// TIA Portal V18 export
// export: Created 2026-06-08T16:32:21.4329296Z, ExportSetting WithDefaults, DisplayName Totally Integrated Automation Portal, DisplayVersion V18, DisplayName TIA Portal Openness, DisplayVersion V18, DisplayName TIA Portal Version Control Interface, DisplayVersion V18, DisplayName STEP 7 Professional, DisplayVersion V18, DisplayName STEP 7 Safety, DisplayVersion V18, DisplayName WinCC Professional, DisplayVersion V18
FUNCTION_BLOCK "Assembly_Blue"   // FB11, LAD
VERSION : 0.1
// stored: AutoNumber true, IsIECCheckEnabled false, UDAEnableTagReadback false
   VAR_TEMP   // added for the SCL form of the ladder/FBD networks
      _w1 : Bool;
      _s5time1 : S5Time;
   END_VAR
BEGIN

REGION Network 1: Clamp when blue lid in place
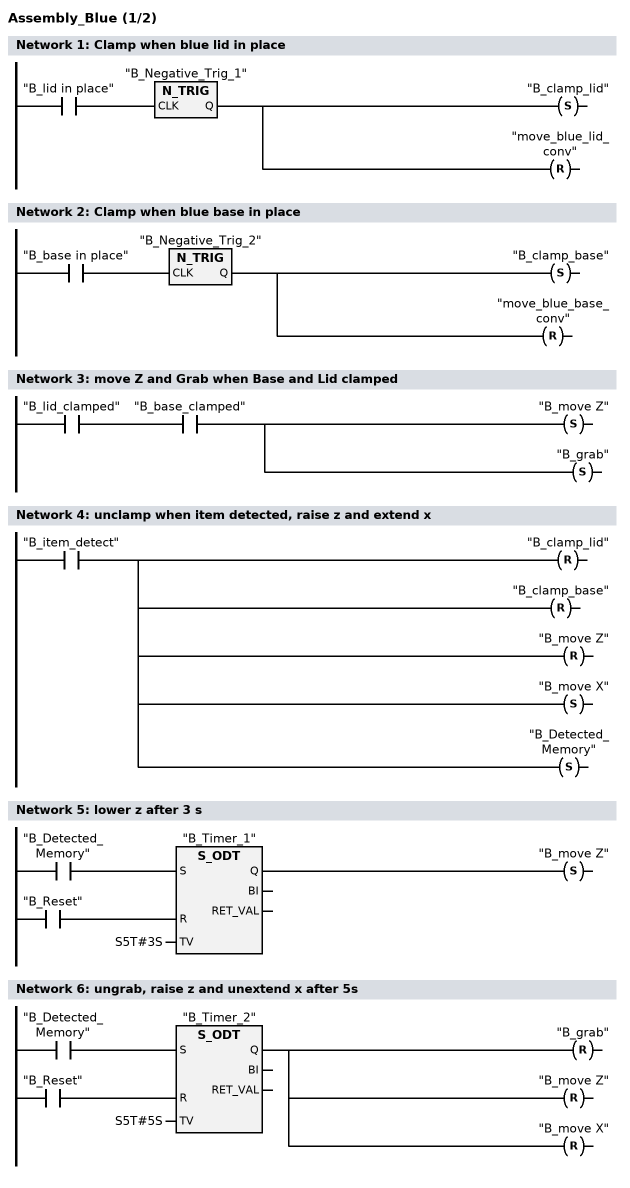
   RUNG wire#powerrail
      Contact( "B_lid in place" )
      N_Trig( "B_Negative_Trig_1" )
      wire#w1
      S_Coil( "B_clamp_lid" )
   END_RUNG
   RUNG wire#w1
      R_Coil( "move_blue_lid_conv" )
   END_RUNG
   // the same network as SCL:
   #_w1 := NOT "B_lid in place" AND "B_Negative_Trig_1";   // falling edge
   "B_Negative_Trig_1" := "B_lid in place";
   IF #_w1 THEN
       "B_clamp_lid" := TRUE;
       "move_blue_lid_conv" := FALSE;
   END_IF;
END_REGION

REGION Network 2: Clamp when blue base in place
   RUNG wire#powerrail
      Contact( "B_base in place" )
      N_Trig( "B_Negative_Trig_2" )
      wire#w1
      S_Coil( "B_clamp_base" )
   END_RUNG
   RUNG wire#w1
      R_Coil( "move_blue_base_conv" )
   END_RUNG
   // the same network as SCL:
   #_w1 := NOT "B_base in place" AND "B_Negative_Trig_2";   // falling edge
   "B_Negative_Trig_2" := "B_base in place";
   IF #_w1 THEN
       "B_clamp_base" := TRUE;
       "move_blue_base_conv" := FALSE;
   END_IF;
END_REGION

REGION Network 3: move Z and Grab when Base and Lid clamped
   RUNG wire#powerrail
      Contact( "B_lid_clamped" )
      Contact( "B_base_clamped" )
      wire#w1
      S_Coil( "B_move Z" )
   END_RUNG
   RUNG wire#w1
      S_Coil( "B_grab" )
   END_RUNG
   // the same network as SCL:
   IF "B_lid_clamped" AND "B_base_clamped" THEN
       "B_move Z" := TRUE;
       "B_grab" := TRUE;
   END_IF;
END_REGION

REGION Network 4: unclamp when item detected, raise z and extend x
   RUNG wire#powerrail
      Contact( "B_item_detect" )
      wire#w1
      R_Coil( "B_clamp_lid" )
   END_RUNG
   RUNG wire#w1
      R_Coil( "B_clamp_base" )
   END_RUNG
   RUNG wire#w1
      R_Coil( "B_move Z" )
   END_RUNG
   RUNG wire#w1
      S_Coil( "B_move X" )
   END_RUNG
   RUNG wire#w1
      S_Coil( "B_Detected_Memory" )
   END_RUNG
   // the same network as SCL:
   IF "B_item_detect" THEN
       "B_clamp_lid" := FALSE;
       "B_clamp_base" := FALSE;
       "B_move Z" := FALSE;
       "B_move X" := TRUE;
       "B_Detected_Memory" := TRUE;
   END_IF;
END_REGION

REGION Network 5: lower z after 3 s
   RUNG wire#powerrail
      Contact( "B_Detected_Memory" )
      S_ODT(T_NO := "B_Timer_1", R := wire#w1, TV := S5T#3S, BI =>, RET_VAL =>)
      S_Coil( "B_move Z" )
   END_RUNG
   RUNG wire#powerrail
      Contact( "B_Reset" )
   END_RUNG wire#w1
   // the same network as SCL:
   #_s5time1 := S_ODT(T_NO := "B_Timer_1", S := "B_Detected_Memory", R := "B_Reset", TV := S5T#3S, Q => #_w1);
   IF #_w1 THEN "B_move Z" := TRUE; END_IF;
END_REGION

REGION Network 6: ungrab, raise z and unextend x after 5s
   RUNG wire#powerrail
      Contact( "B_Detected_Memory" )
      S_ODT(T_NO := "B_Timer_2", R := wire#w1, TV := S5T#5S, BI =>, RET_VAL =>)
      wire#w2
      R_Coil( "B_grab" )
   END_RUNG
   RUNG wire#powerrail
      Contact( "B_Reset" )
   END_RUNG wire#w1
   RUNG wire#w2
      R_Coil( "B_move Z" )
   END_RUNG
   RUNG wire#w2
      R_Coil( "B_move X" )
   END_RUNG
   // the same network as SCL:
   #_s5time1 := S_ODT(T_NO := "B_Timer_2", S := "B_Detected_Memory", R := "B_Reset", TV := S5T#5S, Q => #_w1);
   IF #_w1 THEN
       "B_grab" := FALSE;
       "B_move Z" := FALSE;
       "B_move X" := FALSE;
   END_IF;
END_REGION

REGION Network 7: turn conv on and raise post after 6 s
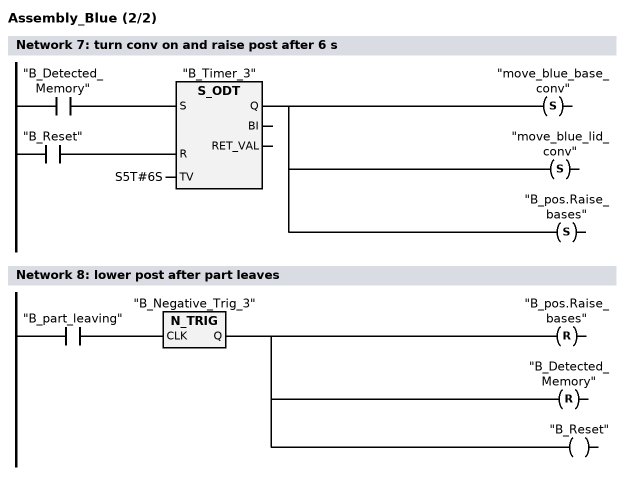
   RUNG wire#powerrail
      Contact( "B_Detected_Memory" )
      S_ODT(T_NO := "B_Timer_3", R := wire#w1, TV := S5T#6S, BI =>, RET_VAL =>)
      wire#w2
      S_Coil( "move_blue_base_conv" )
   END_RUNG
   RUNG wire#powerrail
      Contact( "B_Reset" )
   END_RUNG wire#w1
   RUNG wire#w2
      S_Coil( "move_blue_lid_conv" )
   END_RUNG
   RUNG wire#w2
      S_Coil( "B_pos.Raise_bases" )
   END_RUNG
   // the same network as SCL:
   #_s5time1 := S_ODT(T_NO := "B_Timer_3", S := "B_Detected_Memory", R := "B_Reset", TV := S5T#6S, Q => #_w1);
   IF #_w1 THEN
       "move_blue_base_conv" := TRUE;
       "move_blue_lid_conv" := TRUE;
       "B_pos.Raise_bases" := TRUE;
   END_IF;
END_REGION

REGION Network 8: lower post after part leaves
   RUNG wire#powerrail
      Contact( "B_part_leaving" )
      N_Trig( "B_Negative_Trig_3" )
      wire#w1
      R_Coil( "B_pos.Raise_bases" )
   END_RUNG
   RUNG wire#w1
      R_Coil( "B_Detected_Memory" )
   END_RUNG
   RUNG wire#w1
      Coil( "B_Reset" )
   END_RUNG
   // the same network as SCL:
   #_w1 := NOT "B_part_leaving" AND "B_Negative_Trig_3";   // falling edge
   "B_Negative_Trig_3" := "B_part_leaving";
   IF #_w1 THEN
       "B_pos.Raise_bases" := FALSE;
       "B_Detected_Memory" := FALSE;
   END_IF;
   "B_Reset" := #_w1;
END_REGION
END_FUNCTION_BLOCK
